Yaskawa INFORM job: muffler_cylinder_program.JBI

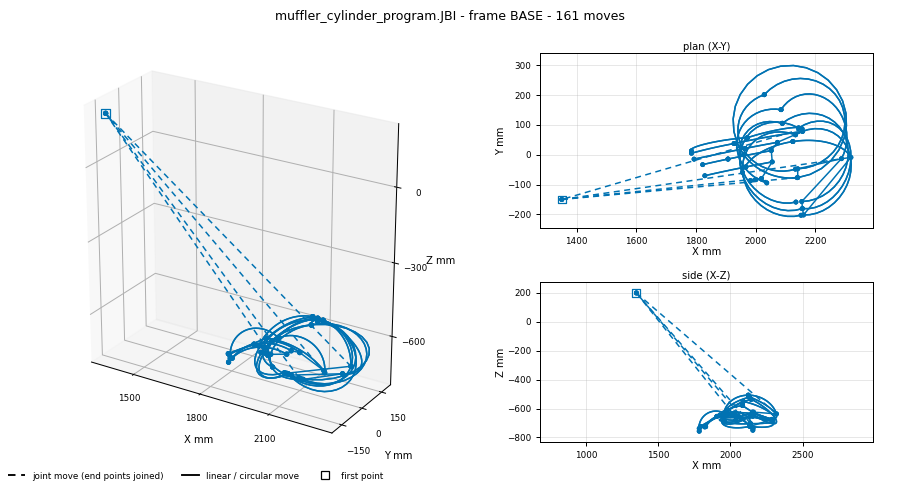
[picture p0: tool path of muffler_cylinder_program.JBI in frame BASE, 161 of 213 moves have a stored position in this frame; points joined in program order, loops and branches not executed]
/JOB
//NAME muffler_cylinder_program
//POS
///NPOS 208,0,208,1,0,2
///TOOL 0
///POSTYPE BASE
///RECTAN
///RCONF 0,0,0,0,0,0,0,0,0,0,0,0,0,0,0,0,0,0,0,0,0,0,0,0
C00000=2319.712,-8.829,-637.166,-175.0000,-81.0987,-165.6741
C00001=2319.712,-8.829,-637.166,-175.0000,-81.0987,-165.6741
C00002=2221.283,44.946,-529.520,175.0000,-43.2325,-129.1574
C00003=2124.955,44.305,-507.577,175.0000,-32.2686,-81.2742
C00004=2124.955,44.305,-507.577,175.0000,-32.2686,-81.2742
C00005=2124.955,44.305,-507.577,175.0000,-32.2686,-81.2742
C00006=2036.278,17.861,-527.858,175.0000,-42.4860,-34.9318
C00007=1956.174,-59.482,-629.877,175.0000,-78.8379,5.0000
C00008=1956.174,-59.482,-629.877,175.0000,-78.8379,5.0000
C00009=1956.174,-59.482,-629.877,175.0000,-78.8379,5.0000
C00010=2036.278,17.861,-527.858,175.0000,-42.4860,-34.9318
C00011=2124.955,44.305,-507.577,175.0000,-32.2686,-81.2742
C00012=2124.955,44.305,-507.577,175.0000,-32.2686,-81.2742
C00013=2124.955,44.305,-507.577,175.0000,-32.2686,-81.2742
C00014=2221.283,44.946,-529.520,175.0000,-43.2325,-129.1574
C00015=2319.712,-8.829,-637.166,-175.0000,-81.0987,-165.6741
C00016=2160.805,-201.906,-624.884,180.0000,-60.0000,98.0702
C00017=2160.805,-201.906,-624.884,180.0000,-60.0000,98.0702
C00018=2305.995,26.906,-625.360,175.0000,-73.1592,-160.3310
C00019=2133.787,67.091,-521.419,-175.0000,-32.4548,-88.2112
C00020=2133.787,67.091,-521.419,-175.0000,-32.4548,-88.2112
C00021=2133.787,67.091,-521.419,-175.0000,-32.4548,-88.2112
C00022=1957.538,-26.114,-625.371,175.0000,-73.1628,-5.0000
C00023=2152.449,-202.906,-624.868,-180.0000,-60.0000,95.2352
C00024=2152.449,-202.906,-624.868,-180.0000,-60.0000,95.2352
C00025=2152.449,-202.906,-624.868,-180.0000,-60.0000,95.2352
C00026=1957.538,-26.114,-625.371,175.0000,-73.1628,-5.0000
C00027=2133.787,67.091,-521.419,-175.0000,-32.4548,-88.2112
C00028=2133.787,67.091,-521.419,-175.0000,-32.4548,-88.2112
C00029=2133.787,67.091,-521.419,-175.0000,-32.4548,-88.2112
C00030=2305.995,26.906,-625.360,175.0000,-73.1592,-160.3310
C00031=2160.805,-201.906,-624.884,180.0000,-60.0000,98.0702
C00032=2157.583,-180.653,-638.457,180.0000,-60.0000,98.0742
C00033=2157.583,-180.653,-638.457,180.0000,-60.0000,98.0742
C00034=2316.776,25.518,-677.720,175.0000,-85.2423,-168.3370
C00035=2144.330,89.682,-536.178,-175.0000,-33.1240,-95.9541
C00036=2144.330,89.682,-536.178,-175.0000,-33.1240,-95.9541
C00037=2144.330,89.682,-536.178,-175.0000,-33.1240,-95.9541
C00038=1947.737,-29.013,-675.195,175.0000,-84.4678,5.1444
C00039=2156.212,-180.843,-638.456,180.0000,-60.0000,97.6079
C00040=2156.212,-180.843,-638.456,180.0000,-60.0000,97.6079
C00041=2156.212,-180.843,-638.456,180.0000,-60.0000,97.6079
C00042=1947.737,-29.013,-675.195,175.0000,-84.4678,5.1444
C00043=2144.330,89.682,-536.178,-175.0000,-33.1240,-95.9541
C00044=2144.330,89.682,-536.178,-175.0000,-33.1240,-95.9541
C00045=2144.330,89.682,-536.178,-175.0000,-33.1240,-95.9541
C00046=2316.776,25.518,-677.720,175.0000,-85.2423,-168.3370
C00047=2157.583,-180.653,-638.457,180.0000,-60.0000,98.0742
C00048=2154.992,-156.852,-653.564,-180.0000,-60.0000,98.4172
C00049=2154.992,-156.852,-653.564,-180.0000,-60.0000,98.4172
C00050=2290.877,79.573,-639.915,175.0000,-68.5916,-157.0167
C00051=2089.538,105.540,-551.295,175.0000,-33.1299,-66.6954
C00052=2089.538,105.540,-551.295,175.0000,-33.1299,-66.6954
C00053=2089.538,105.540,-551.295,175.0000,-33.1299,-66.6954
C00054=1944.812,0.576,-681.168,-175.0000,-81.6571,5.0000
C00055=2135.296,-158.709,-653.497,180.0000,-60.0000,91.7505
C00056=2135.296,-158.709,-653.497,180.0000,-60.0000,91.7505
C00057=2135.296,-158.709,-653.497,180.0000,-60.0000,91.7505
C00058=1944.812,0.576,-681.168,-175.0000,-81.6571,5.0000
C00059=2089.538,105.540,-551.295,175.0000,-33.1299,-66.6954
C00060=2089.538,105.540,-551.295,175.0000,-33.1299,-66.6954
C00061=2089.538,105.540,-551.295,175.0000,-33.1299,-66.6954
C00062=2290.877,79.573,-639.915,175.0000,-68.5916,-157.0167
C00063=2154.992,-156.852,-653.564,-180.0000,-60.0000,98.4172
C00064=2288.024,-13.187,-674.605,180.0000,-60.0000,157.0715
C00065=2288.024,-13.187,-674.605,180.0000,-60.0000,157.0715
C00066=2297.348,110.930,-693.499,175.0000,-76.5238,-162.6465
C00067=2085.441,151.302,-579.808,175.0000,-32.9530,-68.2628
C00068=2085.441,151.302,-579.808,175.0000,-32.9530,-68.2628
C00069=2085.441,151.302,-579.808,175.0000,-32.9530,-68.2628
C00070=1936.913,35.333,-648.369,180.0000,-60.0000,6.4876
C00071=2037.414,-94.336,-679.898,180.0000,-60.0000,60.3662
C00072=2037.414,-94.336,-679.898,180.0000,-60.0000,60.3662
C00073=2037.414,-94.336,-679.898,180.0000,-60.0000,60.3662
C00074=1936.913,35.333,-648.369,180.0000,-60.0000,6.4876
C00075=2085.441,151.302,-579.808,175.0000,-32.9530,-68.2628
C00076=2085.441,151.302,-579.808,175.0000,-32.9530,-68.2628
C00077=2085.441,151.302,-579.808,175.0000,-32.9530,-68.2628
C00078=2297.348,110.930,-693.499,175.0000,-76.5238,-162.6465
C00079=2288.024,-13.187,-674.605,180.0000,-60.0000,157.0715
C00080=2141.297,-47.127,-723.347,180.0000,-60.0000,99.4156
C00081=2141.297,-47.127,-723.347,180.0000,-60.0000,99.4156
C00082=2299.838,118.113,-701.008,180.0000,-60.0000,179.2204
C00083=2029.054,201.504,-631.460,148.3188,-23.2127,13.6717
C00084=2029.054,201.504,-631.460,148.3188,-23.2127,13.6717
C00085=2029.054,201.504,-631.460,148.3188,-23.2127,13.6717
C00086=1948.396,39.540,-707.739,180.0000,-60.0000,26.1663
C00087=2133.605,-48.229,-723.343,180.0000,-60.0000,96.7974
C00088=2133.605,-48.229,-723.343,180.0000,-60.0000,96.7974
C00089=2133.605,-48.229,-723.343,180.0000,-60.0000,96.7974
C00090=1948.396,39.540,-707.739,180.0000,-60.0000,26.1663
C00091=2029.054,201.504,-631.460,148.3188,-23.2127,13.6717
C00092=2029.054,201.504,-631.460,148.3188,-23.2127,13.6717
C00093=2029.054,201.504,-631.460,148.3188,-23.2127,13.6717
C00094=2299.838,118.113,-701.008,180.0000,-60.0000,179.2204
C00095=2141.297,-47.127,-723.347,180.0000,-60.0000,99.4156
C00096=2141.397,-76.681,-704.891,-180.0000,-60.0000,97.9514
C00097=2141.397,-76.681,-704.891,-180.0000,-60.0000,97.9514
C00098=2288.744,33.923,-695.224,180.0000,-60.0000,161.3029
C00099=1960.274,-0.207,-692.050,180.0000,-60.0000,30.2638
C00100=1960.274,-0.207,-692.050,180.0000,-60.0000,30.2638
C00101=1960.274,-0.207,-692.050,180.0000,-60.0000,30.2638
C00102=1983.207,-25.639,-697.442,180.0000,-60.0000,41.0794
C00103=2139.561,-76.930,-704.890,180.0000,-60.0000,97.3271
C00104=2139.561,-76.930,-704.890,180.0000,-60.0000,97.3271
C00105=2139.561,-76.930,-704.890,180.0000,-60.0000,97.3271
C00106=1983.207,-25.639,-697.442,180.0000,-60.0000,41.0794
C00107=1960.274,-0.207,-692.050,180.0000,-60.0000,30.2638
C00108=1960.274,-0.207,-692.050,180.0000,-60.0000,30.2638
C00109=1960.274,-0.207,-692.050,180.0000,-60.0000,30.2638
C00110=2288.744,33.923,-695.224,180.0000,-60.0000,161.3029
C00111=2141.397,-76.681,-704.891,-180.0000,-60.0000,97.9514
C00112=2019.658,-79.422,-638.418,175.0000,6.8392,-5.0000
C00113=2019.658,-79.422,-638.418,175.0000,6.8392,-5.0000
C00114=2008.184,-81.635,-637.286,175.0000,5.0000,-5.0000
C00115=2000.579,-83.113,-636.934,175.0000,5.0000,-5.0000
C00116=2000.579,-83.113,-636.934,175.0000,5.0000,-5.0000
C00117=2000.579,-83.113,-636.934,175.0000,5.0000,-5.0000
C00118=1993.419,-84.513,-636.891,175.0000,-5.0000,5.0000
C00119=1982.245,-86.714,-637.384,175.0000,-5.0000,5.0000
C00120=1982.245,-86.714,-637.384,175.0000,-5.0000,5.0000
C00121=1982.245,-86.714,-637.384,175.0000,-5.0000,5.0000
C00122=1993.419,-84.513,-636.891,175.0000,-5.0000,5.0000
C00123=2000.579,-83.113,-636.934,175.0000,5.0000,-5.0000
C00124=2000.579,-83.113,-636.934,175.0000,5.0000,-5.0000
C00125=2000.579,-83.113,-636.934,175.0000,5.0000,-5.0000
C00126=2008.184,-81.635,-637.286,175.0000,5.0000,-5.0000
C00127=2019.658,-79.422,-638.418,175.0000,6.8392,-5.0000
C00128=2055.809,-23.944,-651.713,173.6074,20.8215,-5.0000
C00129=2055.809,-23.944,-651.713,173.6074,20.8215,-5.0000
C00130=2009.928,-32.573,-639.725,175.0000,6.6760,-5.0000
C00131=1967.170,-40.929,-639.296,175.0000,-6.2094,5.0000
C00132=1967.170,-40.929,-639.296,175.0000,-6.2094,5.0000
C00133=1967.170,-40.929,-639.296,175.0000,-6.2094,5.0000
C00134=1926.434,-49.170,-648.447,-175.0000,-18.7782,-5.0000
C00135=1829.806,-70.357,-726.002,-175.0000,-57.4056,10.0196
C00136=1829.806,-70.357,-726.002,-175.0000,-57.4056,10.0196
C00137=1829.806,-70.357,-726.002,-175.0000,-57.4056,10.0196
C00138=1926.434,-49.170,-648.447,-175.0000,-18.7782,-5.0000
C00139=1967.170,-40.929,-639.296,175.0000,-6.2094,5.0000
C00140=1967.170,-40.929,-639.296,175.0000,-6.2094,5.0000
C00141=1967.170,-40.929,-639.296,175.0000,-6.2094,5.0000
C00142=2009.928,-32.573,-639.725,175.0000,6.6760,-5.0000
C00143=2055.809,-23.944,-651.713,173.6074,20.8215,-5.0000
C00144=2052.687,13.989,-654.540,173.2189,22.1443,-5.0000
C00145=2052.687,13.989,-654.540,173.2189,22.1443,-5.0000
C00146=2009.148,5.842,-641.761,175.0000,8.6423,-5.0000
C00147=1907.476,-14.417,-654.057,-175.0000,-22.5179,-5.0000
C00148=1907.476,-14.417,-654.057,-175.0000,-22.5179,-5.0000
C00149=1907.476,-14.417,-654.057,-175.0000,-22.5179,-5.0000
C00150=1837.763,-29.585,-706.014,175.0000,-49.5036,9.6656
C00151=1822.518,-33.188,-727.113,-175.0000,-57.4132,10.0199
C00152=1822.518,-33.188,-727.113,-175.0000,-57.4132,10.0199
C00153=1822.518,-33.188,-727.113,-175.0000,-57.4132,10.0199
C00154=1837.763,-29.585,-706.014,175.0000,-49.5036,9.6656
C00155=1907.476,-14.417,-654.057,-175.0000,-22.5179,-5.0000
C00156=1907.476,-14.417,-654.057,-175.0000,-22.5179,-5.0000
C00157=1907.476,-14.417,-654.057,-175.0000,-22.5179,-5.0000
C00158=2009.148,5.842,-641.761,175.0000,8.6423,-5.0000
C00159=2052.687,13.989,-654.540,173.2189,22.1443,-5.0000
C00160=2073.325,41.704,-668.468,175.0000,-31.7695,-166.2619
C00161=2073.325,41.704,-668.468,175.0000,-31.7695,-166.2619
C00162=2023.104,32.520,-646.454,175.0000,14.2928,-5.0000
C00163=1964.920,21.313,-640.293,175.0000,-5.0000,5.0000
C00164=1964.920,21.313,-640.293,175.0000,-5.0000,5.0000
C00165=1964.920,21.313,-640.293,175.0000,-5.0000,5.0000
C00166=1845.173,-3.689,-693.662,175.0000,-44.1229,9.3734
C00167=1793.717,-14.687,-723.793,180.0000,-60.0000,10.1380
C00168=1793.717,-14.687,-723.793,180.0000,-60.0000,10.1380
C00169=1793.717,-14.687,-723.793,180.0000,-60.0000,10.1380
C00170=1845.173,-3.689,-693.662,175.0000,-44.1229,9.3734
C00171=1964.920,21.313,-640.293,175.0000,-5.0000,5.0000
C00172=1964.920,21.313,-640.293,175.0000,-5.0000,5.0000
C00173=1964.920,21.313,-640.293,175.0000,-5.0000,5.0000
C00174=2023.104,32.520,-646.454,175.0000,14.2928,-5.0000
C00175=2073.325,41.704,-668.468,175.0000,-31.7695,-166.2619
C00176=2157.476,78.171,-737.096,180.0000,-60.0000,-168.6226
C00177=2157.476,78.171,-737.096,180.0000,-60.0000,-168.6226
C00178=2088.003,67.894,-682.902,175.0000,-38.9331,-166.8840
C00179=1928.043,37.679,-645.660,-175.0000,-13.1864,-5.0000
C00180=1928.043,37.679,-645.660,-175.0000,-13.1864,-5.0000
C00181=1928.043,37.679,-645.660,-175.0000,-13.1864,-5.0000
C00182=1826.591,15.935,-710.009,175.0000,-50.5425,9.7166
C00183=1784.985,5.152,-737.891,180.0000,-60.0000,10.8048
C00184=1784.985,5.152,-737.891,180.0000,-60.0000,10.8048
C00185=1784.985,5.152,-737.891,180.0000,-60.0000,10.8048
C00186=1826.591,15.935,-710.009,175.0000,-50.5425,9.7166
C00187=1928.043,37.679,-645.660,-175.0000,-13.1864,-5.0000
C00188=1928.043,37.679,-645.660,-175.0000,-13.1864,-5.0000
C00189=1928.043,37.679,-645.660,-175.0000,-13.1864,-5.0000
C00190=2088.003,67.894,-682.902,175.0000,-38.9331,-166.8840
C00191=2157.476,78.171,-737.096,180.0000,-60.0000,-168.6226
C00192=2156.103,86.733,-750.155,180.0000,-60.0000,-169.1506
C00193=2156.103,86.733,-750.155,180.0000,-60.0000,-169.1506
C00194=2155.783,88.219,-739.042,180.0000,-60.0000,-168.6925
C00195=1972.258,57.091,-641.031,175.0000,5.0000,-5.0000
C00196=1972.258,57.091,-641.031,175.0000,5.0000,-5.0000
C00197=1972.258,57.091,-641.031,175.0000,5.0000,-5.0000
C00198=1782.962,15.345,-738.363,180.0000,-60.0000,10.8121
C00199=1784.847,13.068,-756.963,180.0000,-60.0000,11.5996
C00200=1784.847,13.068,-756.963,180.0000,-60.0000,11.5996
C00201=1784.847,13.068,-756.963,180.0000,-60.0000,11.5996
C00202=1782.962,15.345,-738.363,180.0000,-60.0000,10.8121
C00203=1972.258,57.091,-641.031,175.0000,5.0000,-5.0000
C00204=1972.258,57.091,-641.031,175.0000,5.0000,-5.0000
C00205=1972.258,57.091,-641.031,175.0000,5.0000,-5.0000
C00206=2155.783,88.219,-739.042,180.0000,-60.0000,-168.6925
C00207=2156.103,86.733,-750.155,180.0000,-60.0000,-169.1506
///POSTYPE PULSE
///PULSE
EC00000=266240
EC00001=266240
EC00002=266240
EC00003=266240
EC00004=266240
EC00005=266240
EC00006=266240
EC00007=266240
EC00008=266240
EC00009=266240
EC00010=266240
EC00011=266240
EC00012=266240
EC00013=266240
EC00014=266240
EC00015=266240
EC00016=266240
EC00017=266240
EC00018=266240
EC00019=266240
EC00020=266240
EC00021=266240
EC00022=266240
EC00023=266240
EC00024=266240
EC00025=266240
EC00026=266240
EC00027=266240
EC00028=266240
EC00029=266240
EC00030=266240
EC00031=266240
EC00032=266240
EC00033=266240
EC00034=266240
EC00035=266240
EC00036=266240
EC00037=266240
EC00038=266240
EC00039=266240
EC00040=266240
EC00041=266240
EC00042=266240
EC00043=266240
EC00044=266240
EC00045=266240
EC00046=266240
EC00047=266240
EC00048=266240
EC00049=266240
EC00050=266240
EC00051=266240
EC00052=266240
EC00053=266240
EC00054=266240
EC00055=266240
EC00056=266240
EC00057=266240
EC00058=266240
EC00059=266240
EC00060=266240
EC00061=266240
EC00062=266240
EC00063=266240
EC00064=266240
EC00065=266240
EC00066=266240
EC00067=266240
EC00068=266240
EC00069=266240
EC00070=266240
EC00071=266240
EC00072=266240
EC00073=266240
EC00074=266240
EC00075=266240
EC00076=266240
EC00077=266240
EC00078=266240
EC00079=266240
EC00080=266240
EC00081=266240
EC00082=266240
EC00083=266240
EC00084=266240
EC00085=266240
EC00086=266240
EC00087=266240
EC00088=266240
EC00089=266240
EC00090=266240
EC00091=266240
EC00092=266240
EC00093=266240
EC00094=266240
EC00095=266240
EC00096=266240
EC00097=266240
EC00098=266240
EC00099=266240
EC00100=266240
EC00101=266240
EC00102=266240
EC00103=266240
EC00104=266240
EC00105=266240
EC00106=266240
EC00107=266240
EC00108=266240
EC00109=266240
EC00110=266240
EC00111=266240
EC00112=282624
EC00113=282624
EC00114=282624
EC00115=282624
EC00116=282624
EC00117=282624
EC00118=282624
EC00119=282624
EC00120=282624
EC00121=282624
EC00122=282624
EC00123=282624
EC00124=282624
EC00125=282624
EC00126=282624
EC00127=282624
EC00128=282624
EC00129=282624
EC00130=282624
EC00131=282624
EC00132=282624
EC00133=282624
EC00134=282624
EC00135=282624
EC00136=282624
EC00137=282624
EC00138=282624
EC00139=282624
EC00140=282624
EC00141=282624
EC00142=282624
EC00143=282624
EC00144=282624
EC00145=282624
EC00146=282624
EC00147=282624
EC00148=282624
EC00149=282624
EC00150=282624
EC00151=282624
EC00152=282624
EC00153=282624
EC00154=282624
EC00155=282624
EC00156=282624
EC00157=282624
EC00158=282624
EC00159=282624
EC00160=282624
EC00161=282624
EC00162=282624
EC00163=282624
EC00164=282624
EC00165=282624
EC00166=282624
EC00167=282624
EC00168=282624
EC00169=282624
EC00170=282624
EC00171=282624
EC00172=282624
EC00173=282624
EC00174=282624
EC00175=282624
EC00176=282624
EC00177=282624
EC00178=282624
EC00179=282624
EC00180=282624
EC00181=282624
EC00182=282624
EC00183=282624
EC00184=282624
EC00185=282624
EC00186=282624
EC00187=282624
EC00188=282624
EC00189=282624
EC00190=282624
EC00191=282624
EC00192=282624
EC00193=282624
EC00194=282624
EC00195=282624
EC00196=282624
EC00197=282624
EC00198=282624
EC00199=282624
EC00200=282624
EC00201=282624
EC00202=282624
EC00203=282624
EC00204=282624
EC00205=282624
EC00206=282624
EC00207=282624
///POSTYPE BASE
///RECTAN
///RCONF 1,0,0,0,0,0,0,0,0,0,0,0,0,0,0,0,0,0,0,0,0,0,0,0
P00009=1350.000,-150.000,200.000,-180.0000,-45.0000,0.0000
///POSTYPE PULSE
///PULSE
EX00000=0
EX00001=282624
//INST
///DATE 2023/08/13 12:16
///ATTR SC,RW,RJ
////FRAME BASE
///GROUP1 RB1,ST1
NOP
MOVJ P009 EX000 VJ=15.00
MOVJ C00000 EC00000 VJ=15.00
CALL JOB:SPYON
MOVC C00001 EC00001 V=150.0
MOVC C00002 EC00002 V=150.0
MOVC C00003 EC00003 V=150.0
MOVL C00004 EC00004 V=150.0
MOVC C00005 EC00005 V=150.0
MOVC C00006 EC00006 V=150.0
MOVC C00007 EC00007 V=150.0
MOVL C00008 EC00008 V=150.0
MOVC C00009 EC00009 V=150.0
MOVC C00010 EC00010 V=150.0
MOVC C00011 EC00011 V=150.0
MOVL C00012 EC00012 V=150.0
MOVC C00013 EC00013 V=150.0
MOVC C00014 EC00014 V=150.0
MOVC C00015 EC00015 V=150.0
MOVL C00016 EC00016 V=150.0
MOVC C00017 EC00017 V=150.0
MOVC C00018 EC00018 V=150.0
MOVC C00019 EC00019 V=150.0
MOVL C00020 EC00020 V=150.0
MOVC C00021 EC00021 V=150.0
MOVC C00022 EC00022 V=150.0
MOVC C00023 EC00023 V=150.0
MOVL C00024 EC00024 V=150.0
MOVC C00025 EC00025 V=150.0
MOVC C00026 EC00026 V=150.0
MOVC C00027 EC00027 V=150.0
MOVL C00028 EC00028 V=150.0
MOVC C00029 EC00029 V=150.0
MOVC C00030 EC00030 V=150.0
MOVC C00031 EC00031 V=150.0
MOVL C00032 EC00032 V=150.0
MOVC C00033 EC00033 V=150.0
MOVC C00034 EC00034 V=150.0
MOVC C00035 EC00035 V=150.0
MOVL C00036 EC00036 V=150.0
MOVC C00037 EC00037 V=150.0
MOVC C00038 EC00038 V=150.0
MOVC C00039 EC00039 V=150.0
MOVL C00040 EC00040 V=150.0
MOVC C00041 EC00041 V=150.0
MOVC C00042 EC00042 V=150.0
MOVC C00043 EC00043 V=150.0
MOVL C00044 EC00044 V=150.0
MOVC C00045 EC00045 V=150.0
MOVC C00046 EC00046 V=150.0
MOVC C00047 EC00047 V=150.0
MOVL C00048 EC00048 V=150.0
MOVC C00049 EC00049 V=150.0
MOVC C00050 EC00050 V=150.0
MOVC C00051 EC00051 V=150.0
MOVL C00052 EC00052 V=150.0
MOVC C00053 EC00053 V=150.0
MOVC C00054 EC00054 V=150.0
MOVC C00055 EC00055 V=150.0
MOVL C00056 EC00056 V=150.0
MOVC C00057 EC00057 V=150.0
MOVC C00058 EC00058 V=150.0
MOVC C00059 EC00059 V=150.0
MOVL C00060 EC00060 V=150.0
MOVC C00061 EC00061 V=150.0
MOVC C00062 EC00062 V=150.0
MOVC C00063 EC00063 V=150.0
MOVL C00064 EC00064 V=150.0
MOVC C00065 EC00065 V=150.0
MOVC C00066 EC00066 V=150.0
MOVC C00067 EC00067 V=150.0
MOVL C00068 EC00068 V=150.0
MOVC C00069 EC00069 V=150.0
MOVC C00070 EC00070 V=150.0
MOVC C00071 EC00071 V=150.0
MOVL C00072 EC00072 V=150.0
MOVC C00073 EC00073 V=150.0
MOVC C00074 EC00074 V=150.0
MOVC C00075 EC00075 V=150.0
MOVL C00076 EC00076 V=150.0
MOVC C00077 EC00077 V=150.0
MOVC C00078 EC00078 V=150.0
MOVC C00079 EC00079 V=150.0
MOVL C00080 EC00080 V=150.0
MOVC C00081 EC00081 V=150.0
MOVC C00082 EC00082 V=150.0
MOVC C00083 EC00083 V=150.0
MOVL C00084 EC00084 V=150.0
MOVC C00085 EC00085 V=150.0
MOVC C00086 EC00086 V=150.0
MOVC C00087 EC00087 V=150.0
MOVL C00088 EC00088 V=150.0
MOVC C00089 EC00089 V=150.0
MOVC C00090 EC00090 V=150.0
MOVC C00091 EC00091 V=150.0
MOVL C00092 EC00092 V=150.0
MOVC C00093 EC00093 V=150.0
MOVC C00094 EC00094 V=150.0
MOVC C00095 EC00095 V=150.0
MOVL C00096 EC00096 V=150.0
MOVC C00097 EC00097 V=150.0
MOVC C00098 EC00098 V=150.0
MOVC C00099 EC00099 V=150.0
MOVL C00100 EC00100 V=150.0
MOVC C00101 EC00101 V=150.0
MOVC C00102 EC00102 V=150.0
MOVC C00103 EC00103 V=150.0
MOVL C00104 EC00104 V=150.0
MOVC C00105 EC00105 V=150.0
MOVC C00106 EC00106 V=150.0
MOVC C00107 EC00107 V=150.0
MOVL C00108 EC00108 V=150.0
MOVC C00109 EC00109 V=150.0
MOVC C00110 EC00110 V=150.0
MOVC C00111 EC00111 V=150.0
CALL JOB:SPYOF
MOVJ P009 VJ=15.00
MOVL P009 EX000 V=150.0
MOVJ C00112 EC00112 VJ=15.00
CALL JOB:SPYON
MOVC C00113 EC00113 V=150.0
MOVC C00114 EC00114 V=150.0
MOVC C00115 EC00115 V=150.0
MOVL C00116 EC00116 V=150.0
MOVC C00117 EC00117 V=150.0
MOVC C00118 EC00118 V=150.0
MOVC C00119 EC00119 V=150.0
MOVL C00120 EC00120 V=150.0
MOVC C00121 EC00121 V=150.0
MOVC C00122 EC00122 V=150.0
MOVC C00123 EC00123 V=150.0
MOVL C00124 EC00124 V=150.0
MOVC C00125 EC00125 V=150.0
MOVC C00126 EC00126 V=150.0
MOVC C00127 EC00127 V=150.0
MOVL C00128 EC00128 V=150.0
MOVC C00129 EC00129 V=150.0
MOVC C00130 EC00130 V=150.0
MOVC C00131 EC00131 V=150.0
MOVL C00132 EC00132 V=150.0
MOVC C00133 EC00133 V=150.0
MOVC C00134 EC00134 V=150.0
MOVC C00135 EC00135 V=150.0
MOVL C00136 EC00136 V=150.0
MOVC C00137 EC00137 V=150.0
MOVC C00138 EC00138 V=150.0
MOVC C00139 EC00139 V=150.0
MOVL C00140 EC00140 V=150.0
MOVC C00141 EC00141 V=150.0
MOVC C00142 EC00142 V=150.0
MOVC C00143 EC00143 V=150.0
MOVL C00144 EC00144 V=150.0
MOVC C00145 EC00145 V=150.0
MOVC C00146 EC00146 V=150.0
MOVC C00147 EC00147 V=150.0
MOVL C00148 EC00148 V=150.0
MOVC C00149 EC00149 V=150.0
MOVC C00150 EC00150 V=150.0
MOVC C00151 EC00151 V=150.0
MOVL C00152 EC00152 V=150.0
MOVC C00153 EC00153 V=150.0
MOVC C00154 EC00154 V=150.0
MOVC C00155 EC00155 V=150.0
MOVL C00156 EC00156 V=150.0
MOVC C00157 EC00157 V=150.0
MOVC C00158 EC00158 V=150.0
MOVC C00159 EC00159 V=150.0
MOVL C00160 EC00160 V=150.0
MOVC C00161 EC00161 V=150.0
MOVC C00162 EC00162 V=150.0
MOVC C00163 EC00163 V=150.0
MOVL C00164 EC00164 V=150.0
MOVC C00165 EC00165 V=150.0
MOVC C00166 EC00166 V=150.0
MOVC C00167 EC00167 V=150.0
MOVL C00168 EC00168 V=150.0
MOVC C00169 EC00169 V=150.0
MOVC C00170 EC00170 V=150.0
MOVC C00171 EC00171 V=150.0
MOVL C00172 EC00172 V=150.0
MOVC C00173 EC00173 V=150.0
MOVC C00174 EC00174 V=150.0
MOVC C00175 EC00175 V=150.0
MOVL C00176 EC00176 V=150.0
MOVC C00177 EC00177 V=150.0
MOVC C00178 EC00178 V=150.0
MOVC C00179 EC00179 V=150.0
MOVL C00180 EC00180 V=150.0
MOVC C00181 EC00181 V=150.0
MOVC C00182 EC00182 V=150.0
MOVC C00183 EC00183 V=150.0
MOVL C00184 EC00184 V=150.0
MOVC C00185 EC00185 V=150.0
MOVC C00186 EC00186 V=150.0
MOVC C00187 EC00187 V=150.0
MOVL C00188 EC00188 V=150.0
MOVC C00189 EC00189 V=150.0
MOVC C00190 EC00190 V=150.0
MOVC C00191 EC00191 V=150.0
MOVL C00192 EC00192 V=150.0
MOVC C00193 EC00193 V=150.0
MOVC C00194 EC00194 V=150.0
MOVC C00195 EC00195 V=150.0
MOVL C00196 EC00196 V=150.0
MOVC C00197 EC00197 V=150.0
MOVC C00198 EC00198 V=150.0
MOVC C00199 EC00199 V=150.0
MOVL C00200 EC00200 V=150.0
MOVC C00201 EC00201 V=150.0
MOVC C00202 EC00202 V=150.0
MOVC C00203 EC00203 V=150.0
MOVL C00204 EC00204 V=150.0
MOVC C00205 EC00205 V=150.0
MOVC C00206 EC00206 V=150.0
MOVC C00207 EC00207 V=150.0
CALL JOB:SPYOF
MOVJ P009 VJ=15.00
MOVL P009 EX001 V=150.0
END
